Xinje XDPPro project, PLC1: XD5-48T6 (software 3.5.3 2018-11-19)

PROGRAM Ladder

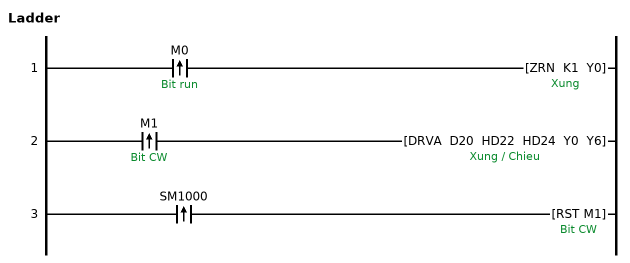
LDP    M0	; Bit run
ZRN    K1 Y0	; Xung
LDP    M1	; Bit CW
DRVA   D20 HD22 HD24 Y0 Y6	; Xung / Chieu
LDP    SM1000
RST    M1	; Bit CW

COMMENTS (devices not used above)
M2	Bit CCW
HD0	So xung
HD2	Tan so
HD4	Gia toc
HD10	Khoang cach (mm)